// Mitsubishi GX Works2 project: 실린더제어 abbacc   PLC: Q02/Q02H

PROGRAM MAIN
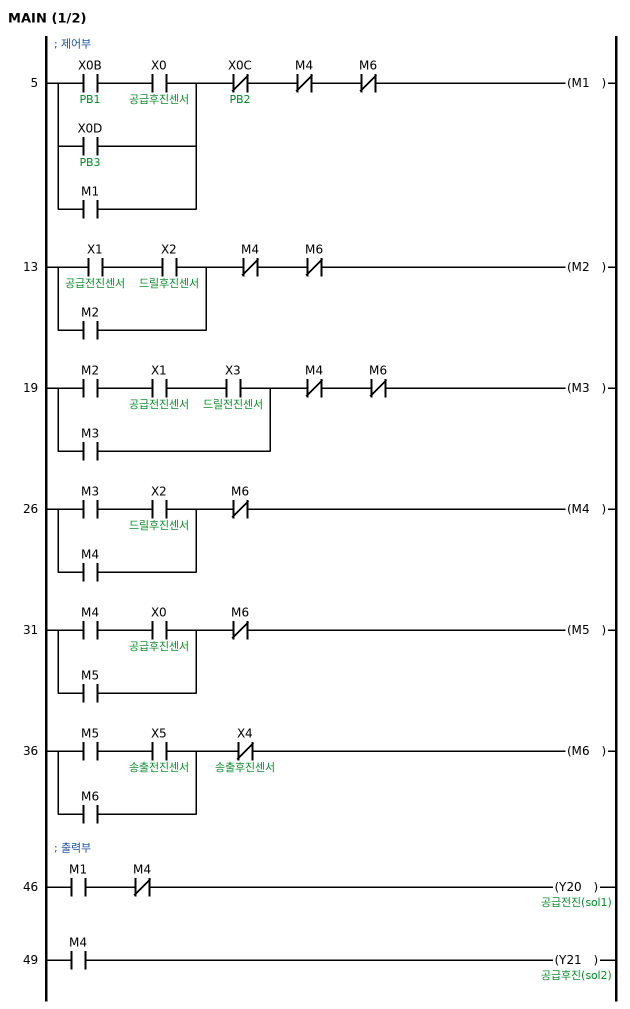
; 제어부
5     LD      X0B  ; PB1
      AND     X0  ; 공급후진센서
      OR      X0D  ; PB3
      OR      M1
      ANI     X0C  ; PB2
      ANI     M4
      ANI     M6
      OUT     M1
13    LD      X1  ; 공급전진센서
      AND     X2  ; 드릴후진센서
      OR      M2
      ANI     M4
      ANI     M6
      OUT     M2
19    LD      M2
      AND     X1  ; 공급전진센서
      AND     X3  ; 드릴전진센서
      OR      M3
      ANI     M4
      ANI     M6
      OUT     M3
26    LD      M3
      AND     X2  ; 드릴후진센서
      OR      M4
      ANI     M6
      OUT     M4
31    LD      M4
      AND     X0  ; 공급후진센서
      OR      M5
      ANI     M6
      OUT     M5
36    LD      M5
      AND     X5  ; 송출전진센서
      OR      M6
      ANI     X4  ; 송출후진센서
      OUT     M6
; 출력부
46    LD      M1
      ANI     M4
      OUT     Y20  ; 공급전진(sol1)
49    LD      M4
      OUT     Y21  ; 공급후진(sol2)
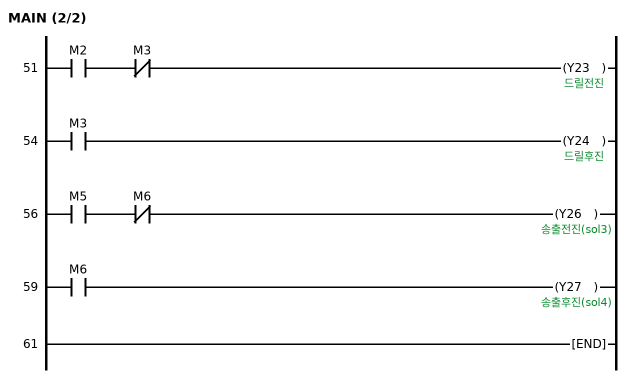
51    LD      M2
      ANI     M3
      OUT     Y23  ; 드릴전진
54    LD      M3
      OUT     Y24  ; 드릴후진
56    LD      M5
      ANI     M6
      OUT     Y26  ; 송출전진(sol3)
59    LD      M6
      OUT     Y27  ; 송출후진(sol4)
61    END
END_PROGRAM
